PROGRAM MAIN
VAR
	fbAdsConnector : AdsConnector;
END_VAR

fbAdsConnector();
fbAdsConnector.Execute();

END_PROGRAM

(* stored: Version 1.1.0.1, ProductVersion 3.1.4024.0
   POU MAIN: Id {a86c6d0f-1010-44d2-ba7b-37cc6bac563a}, SpecialFunc None *)
